// One passing test; used by PRG_TEST_SEQUENCE for the N=1 sequential check.
FUNCTION_BLOCK FB_SequentialSingleSuite EXTENDS TcUnit.FB_TestSuite

TEST('Test_SingleSequentialPass');
AssertTrue(Condition := TRUE, Message := 'Single-suite sequential run');
TEST_FINISHED();

END_FUNCTION_BLOCK

(* stored: Version 1.1.0.1
   POU FB_SequentialSingleSuite: Id {c9861766-2402-41df-8a74-0fbae6a71719}, SpecialFunc None *)
